Omron Sysmac Studio project MODBUS_TPC_CLIENT_NX1P2_plc_s7-1200 (Sysmac Studio 1.45.1.64010, StandardProject)

# Controller new_Controller_0: NX1P2-9024DT version 1.40
Units and slaves: Node86 : NX-ECC201 (E001); Unit 1 : NX-OD5121 (N1); Unit 2 : NX-OD4256 (N2); Unit 3 : NX-ID5342 (N3); Unit 4 : NX-ID5442 (N4); Node1 : GX-ID1611+OD16 (E002)
Task PrimaryTask (priority 4, period or condition 2000): Program0
Library OEN_Communication_V1_0_22 1.0.22 (contents left out)

VAR_GLOBAL
    NX1P2_OUT_0 : BOOL;  (* NX1P2_OUT; at BuiltInIO://cpu/#0/Output_Bit_00 *)
    NX1P2_OUT_1 : BOOL;  (* NX1P2_OUT; at BuiltInIO://cpu/#0/Output_Bit_01 *)
    NX1P2_OUT_2 : BOOL;  (* NX1P2_OUT; at BuiltInIO://cpu/#0/Output_Bit_02 *)
    NX1P2_OUT_3 : BOOL;  (* NX1P2_OUT; at BuiltInIO://cpu/#0/Output_Bit_03 *)
    NX1P2_OUT_4 : BOOL;  (* NX1P2_OUT; at BuiltInIO://cpu/#0/Output_Bit_04 *)
    NX1P2_OUT_5 : BOOL;  (* NX1P2_OUT; at BuiltInIO://cpu/#0/Output_Bit_05 *)
    NX1P2_OUT_6 : BOOL;  (* NX1P2_OUT; at BuiltInIO://cpu/#0/Output_Bit_06 *)
    NX1P2_OUT_7 : BOOL;  (* NX1P2_OUT; at BuiltInIO://cpu/#0/Output_Bit_07 *)
    NX1P2_OUT_8 : BOOL;  (* NX1P2_OUT; at BuiltInIO://cpu/#0/Output_Bit_08 *)
    NX1P2_OUT_9 : BOOL;  (* NX1P2_OUT; at BuiltInIO://cpu/#0/Output_Bit_09 *)
    GX_OUT_0 : BOOL;  (* OD_1611_DT; at ECAT://node#1/Write output 1st word/Out Bit00 *)
    GX_OUT_1 : BOOL;  (* OD_1611_DT; at ECAT://node#1/Write output 1st word/Out Bit01 *)
    GX_OUT_2 : BOOL;  (* OD_1611_DT; at ECAT://node#1/Write output 1st word/Out Bit02 *)
    GX_OUT_3 : BOOL;  (* OD_1611_DT; at ECAT://node#1/Write output 1st word/Out Bit03 *)
    GX_OUT_4 : BOOL;  (* OD_1611_DT; at ECAT://node#1/Write output 1st word/Out Bit04 *)
    GX_OUT_5 : BOOL;  (* OD_1611_DT; at ECAT://node#1/Write output 1st word/Out Bit05 *)
    GX_OUT_6 : BOOL;  (* OD_1611_DT; at ECAT://node#1/Write output 1st word/Out Bit06 *)
    GX_OUT_7 : BOOL;  (* OD_1611_DT; at ECAT://node#1/Write output 1st word/Out Bit07 *)
    GX_OUT_8 : BOOL;  (* OD_1611_DT; at ECAT://node#1/Write output 1st word/Out Bit08 *)
    GX_OUT_9 : BOOL;  (* OD_1611_DT; at ECAT://node#1/Write output 1st word/Out Bit09 *)
    GX_OUT_10 : BOOL;  (* OD_1611_DT; at ECAT://node#1/Write output 1st word/Out Bit10 *)
    GX_OUT_11 : BOOL;  (* OD_1611_DT; at ECAT://node#1/Write output 1st word/Out Bit11 *)
    GX_OUT_12 : BOOL;  (* OD_1611_DT; at ECAT://node#1/Write output 1st word/Out Bit12 *)
    GX_OUT_13 : BOOL;  (* OD_1611_DT; at ECAT://node#1/Write output 1st word/Out Bit13 *)
    GX_OUT_14 : BOOL;  (* OD_1611_DT; at ECAT://node#1/Write output 1st word/Out Bit14 *)
    GX_OUT_15 : BOOL;  (* OD_1611_DT; at ECAT://node#1/Write output 1st word/Out Bit15 *)
    REGISTER_GX_OUT : WORD;  (* OD_1611_DT; at ECAT://node#1/Write output 1st word *)
    NX1P2_IN_0 : BOOL;  (* input_nx1p2_9024dt; at BuiltInIO://cpu/#0/Input_Bit_00 *)
    NX1P2_IN_1 : BOOL;  (* input_nx1p2_9024dt; at BuiltInIO://cpu/#0/Input_Bit_01 *)
    NX1P2_IN_2 : BOOL;  (* input_nx1p2_9024dt; at BuiltInIO://cpu/#0/Input_Bit_02 *)
    NX1P2_IN_3 : BOOL;  (* input_nx1p2_9024dt; at BuiltInIO://cpu/#0/Input_Bit_03 *)
    NX1P2_IN_4 : BOOL;  (* input_nx1p2_9024dt; at BuiltInIO://cpu/#0/Input_Bit_04 *)
    NX1P2_IN_5 : BOOL;  (* input_nx1p2_9024dt; at BuiltInIO://cpu/#0/Input_Bit_05 *)
    NX1P2_IN_6 : BOOL;  (* input_nx1p2_9024dt; at BuiltInIO://cpu/#0/Input_Bit_06 *)
    NX1P2_IN_7 : BOOL;  (* input_nx1p2_9024dt; at BuiltInIO://cpu/#0/Input_Bit_07 *)
    NX1P2_IN_8 : BOOL;  (* input_nx1p2_9024dt; at BuiltInIO://cpu/#0/Input_Bit_08 *)
    NX1P2_IN_9 : BOOL;  (* input_nx1p2_9024dt; at BuiltInIO://cpu/#0/Input_Bit_09 *)
    NX1P2_IN_10 : BOOL;  (* input_nx1p2_9024dt; at BuiltInIO://cpu/#0/Input_Bit_10 *)
    NX1P2_IN_11 : BOOL;  (* input_nx1p2_9024dt; at BuiltInIO://cpu/#0/Input_Bit_11 *)
    NX1P2_IN_12 : BOOL;  (* input_nx1p2_9024dt; at BuiltInIO://cpu/#0/Input_Bit_12 *)
    NX1P2_IN_13 : BOOL;  (* input_nx1p2_9024dt; at BuiltInIO://cpu/#0/Input_Bit_13 *)
    IN_GX_0 : BOOL;  (* INPUT_ID1611; at ECAT://node#1/Read input 1st word/In Bit00 *)
    IN_GX_1 : BOOL;  (* INPUT_ID1611; at ECAT://node#1/Read input 1st word/In Bit01 *)
    IN_GX_2 : BOOL;  (* INPUT_ID1611; at ECAT://node#1/Read input 1st word/In Bit02 *)
    IN_GX_3 : BOOL;  (* INPUT_ID1611; at ECAT://node#1/Read input 1st word/In Bit03 *)
    IN_GX_4 : BOOL;  (* INPUT_ID1611; at ECAT://node#1/Read input 1st word/In Bit04 *)
    IN_GX_5 : BOOL;  (* INPUT_ID1611; at ECAT://node#1/Read input 1st word/In Bit05 *)
    IN_GX_6 : BOOL;  (* INPUT_ID1611; at ECAT://node#1/Read input 1st word/In Bit06 *)
    IN_GX_7 : BOOL;  (* INPUT_ID1611; at ECAT://node#1/Read input 1st word/In Bit07 *)
    IN_GX_8 : BOOL;  (* INPUT_ID1611; at ECAT://node#1/Read input 1st word/In Bit08 *)
    IN_GX_9 : BOOL;  (* INPUT_ID1611; at ECAT://node#1/Read input 1st word/In Bit09 *)
    IN_GX_10 : BOOL;  (* INPUT_ID1611; at ECAT://node#1/Read input 1st word/In Bit10 *)
    IN_GX_11 : BOOL;  (* INPUT_ID1611; at ECAT://node#1/Read input 1st word/In Bit11 *)
    IN_GX_12 : BOOL;  (* INPUT_ID1611; at ECAT://node#1/Read input 1st word/In Bit12 *)
    IN_GX_13 : BOOL;  (* INPUT_ID1611; at ECAT://node#1/Read input 1st word/In Bit13 *)
    IN_GX_14 : BOOL;  (* INPUT_ID1611; at ECAT://node#1/Read input 1st word/In Bit14 *)
    IN_GX_15 : BOOL;  (* INPUT_ID1611; at ECAT://node#1/Read input 1st word/In Bit15 *)
    REGISTER_IN_GX : WORD;  (* INPUT_ID1611; at ECAT://node#1/Read input 1st word *)
    ERROR_GX : BYTE;  (* INPUT_ID1611; at ECAT://node#1/Sysmac Error Status *)
END_VAR
VAR_GLOBAL RETAIN
    D0 AT %D0 : INT;
    D1 AT %D1 : INT;
    D2 AT %D2 : INT;
    D3 AT %D3 : INT;
END_VAR
VAR_GLOBAL
    W0 AT %W0 : INT;
END_VAR

PROGRAM Program0
VAR
    DISCONNECT_TCP_CLIENT : BOOL;
    TCP_CLIENT_CONNECT : BOOL;
    T_CONNECT_TCP : TON;
    T_CONNECT_TCP_CLIENT : TON;
    MODBUS_CLIENT : OEN\Modbus\ModbusTCP_Client;
    REQUEST_CLIENT : ARRAY[0..3] OF OEN\Modbus\sModbusReq := [(Enable := True, NodeAdr := 0, FunctionCode := Fn03_ReadHoldingRegisters, Read := (StartAddressRemote := 0, StartAddressLocal := 0, Count := 4), Write := (StartAddressRemote := 0, StartAddressLocal := 0, Count := 0)), (Enable := True, NodeAdr := 0, FunctionCode := Fn16_WriteMultipleRegisters, Read := (StartAddressRemote := 0, StartAddressLocal := 0, Count := 0), Write := (StartAddressRemote := 4, StartAddressLocal := 4, Count := 6)), (Enable := True, NodeAdr := 0, FunctionCode := Fn03_ReadHoldingRegisters, Read := (StartAddressRemote := 10, StartAddressLocal := 10, Count := 6), Write := (StartAddressRemote := 0, StartAddressLocal := 0, Count := 0)), (Enable := True, NodeAdr := 0, FunctionCode := Fn16_WriteMultipleRegisters, Read := (StartAddressRemote := 0, StartAddressLocal := 0, Count := 0), Write := (StartAddressRemote := 17, StartAddressLocal := 17, Count := 6))];
    DATA_COIL_CLIENT : ARRAY[0..16] OF BOOL;
    DISCRETELINPUT_CLIENT : ARRAY[0..16] OF BOOL;
    INPUT_REGISTER_CLIENT : ARRAY[0..16] OF WORD;
    HOLDINGREGISTERR_CLIENT : ARRAY[0..31] OF WORD;
    REQUEST_DONE : BOOL;
    REQUEST_CLYCLE_TIME : TIME;
    TCP_CONNECT : BOOL;
    DATA_WRITE_0 : WORD;
    DATA_WRITE_1 : WORD;
    DATA_WRITE_2 : WORD;
    DATA_WRITE_3 : WORD;
    DATA_WRITE_4 AT %W0 : WORD;
    DATA_WRITE_5 : WORD;
    INT_DATA_WRITE_5 : INT;
    INT_WRITE_4 : INT;
    DINT_DATA_WRITE_6 : DINT;
    INT_DATA_READ_4 : INT;
    INT_DATA_READ_0 : INT;
    INT_DATA_READ_1 : DINT;
    INT_DATA_READ_5 : INT;
    INT_DATA_READ_6 : INT;
    INT_DATA_LOW_READ_5 : INT;
    INT_DATA_HIGH_READ_5 : INT;
    INT_DATA_READ_7 : INT;
    DISCONNECT_MODBUS_TCP_CLIENT : BOOL;
    VAL_CONTROL_OD1611 : DWORD;
    VAL_TRGIAN_RES_01 : WORD;
    INT_DATA_CONTROL : DINT;
    INT_HIGH_RES_DWORD_0 : DINT;
    OUT : BOOL;
    DATA_READ_12 : WORD;
    DATA_READ_13 : WORD;
    REGISTER_12 : DINT;
    T_COUNT_1 : TON;
    DATA_READ_4 : WORD;
    COUNT_1 : INT;
END_VAR
VAR RETAIN
    SV_COUNT_1 : int;
END_VAR
VAR
    T_COUNT_2 : TON;
    H : INT;
END_VAR
VAR RETAIN
    DATA_RES_15 AT %D15 : WORD;
END_VAR
VAR
    T1 : TON;
    T2 : TON;
END_VAR
VAR_EXTERNAL
    REGISTER_GX_OUT : WORD;
    NX1P2_IN_0 : BOOL;
    IN_GX_0 : BOOL;
    NX1P2_OUT_3 : BOOL;
    IN_GX_1 : BOOL;
    IN_GX_2 : BOOL;
    D0 : INT;
    IN_GX_3 : BOOL;
    D1 : INT;
    IN_GX_4 : BOOL;
    D2 : INT;
    D3 : INT;
    NX1P2_OUT_5 : BOOL;
    IN_GX_6 : BOOL;
END_VAR
VAR
    _e1 : R_TRIG;
    _e2 : R_TRIG;
    _e3 : R_TRIG;
    _e4 : R_TRIG;
    _e5 : R_TRIG;
    _e6 : R_TRIG;
    _e7 : R_TRIG;
END_VAR

(* Section modbus_tcp_client: ladder, written here as Structured Text *)

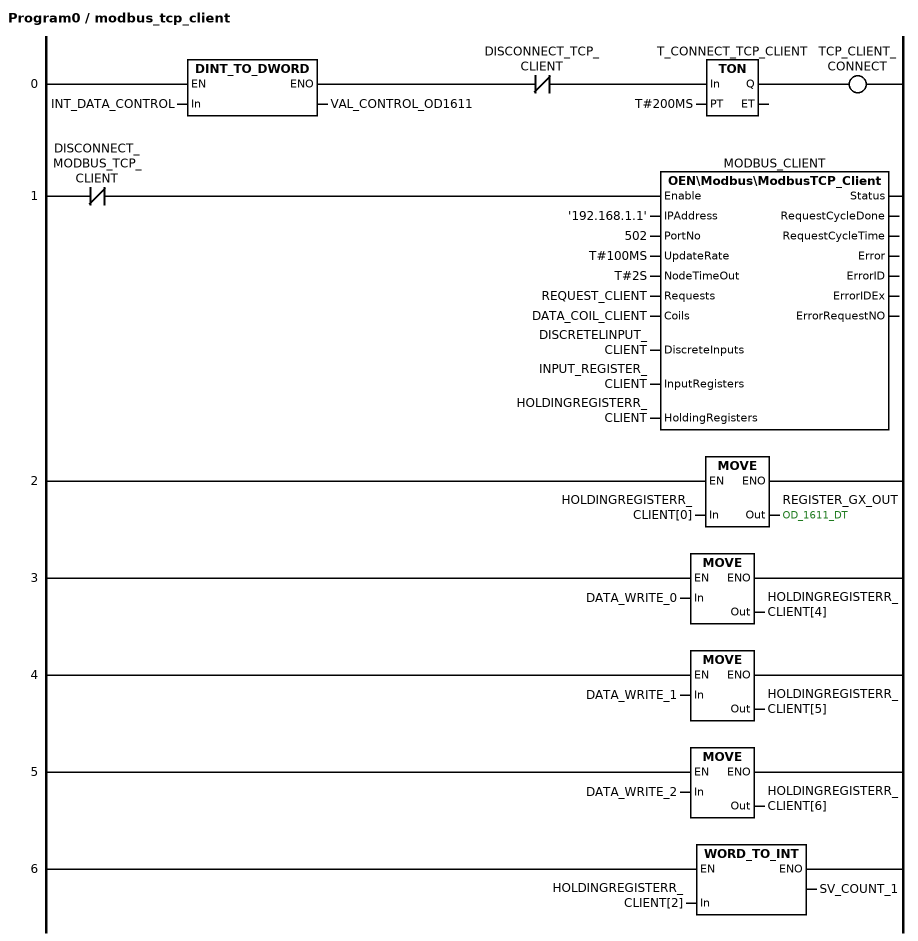
(* Rung 0 *)
VAL_CONTROL_OD1611 := DINT_TO_DWORD(In := INT_DATA_CONTROL);
T_CONNECT_TCP_CLIENT(In := NOT DISCONNECT_TCP_CLIENT, PT := T#200MS);
TCP_CLIENT_CONNECT := T_CONNECT_TCP_CLIENT.Q;
(* Rung 1 *)
MODBUS_CLIENT(Enable := NOT DISCONNECT_MODBUS_TCP_CLIENT, IPAddress := '192.168.1.1', PortNo := 502, UpdateRate := T#100MS, NodeTimeOut := T#2S, Requests := REQUEST_CLIENT, Coils := DATA_COIL_CLIENT, DiscreteInputs := DISCRETELINPUT_CLIENT, InputRegisters := INPUT_REGISTER_CLIENT, HoldingRegisters := HOLDINGREGISTERR_CLIENT);
(* Rung 2 *)
REGISTER_GX_OUT := HOLDINGREGISTERR_CLIENT[0];
(* Rung 3 *)
HOLDINGREGISTERR_CLIENT[4] := DATA_WRITE_0;
(* Rung 4 *)
HOLDINGREGISTERR_CLIENT[5] := DATA_WRITE_1;
(* Rung 5 *)
HOLDINGREGISTERR_CLIENT[6] := DATA_WRITE_2;
(* Rung 6 *)
SV_COUNT_1 := WORD_TO_INT(In := HOLDINGREGISTERR_CLIENT[2]);

(* Section write_data_res_4_10: ladder, written here as Structured Text *)

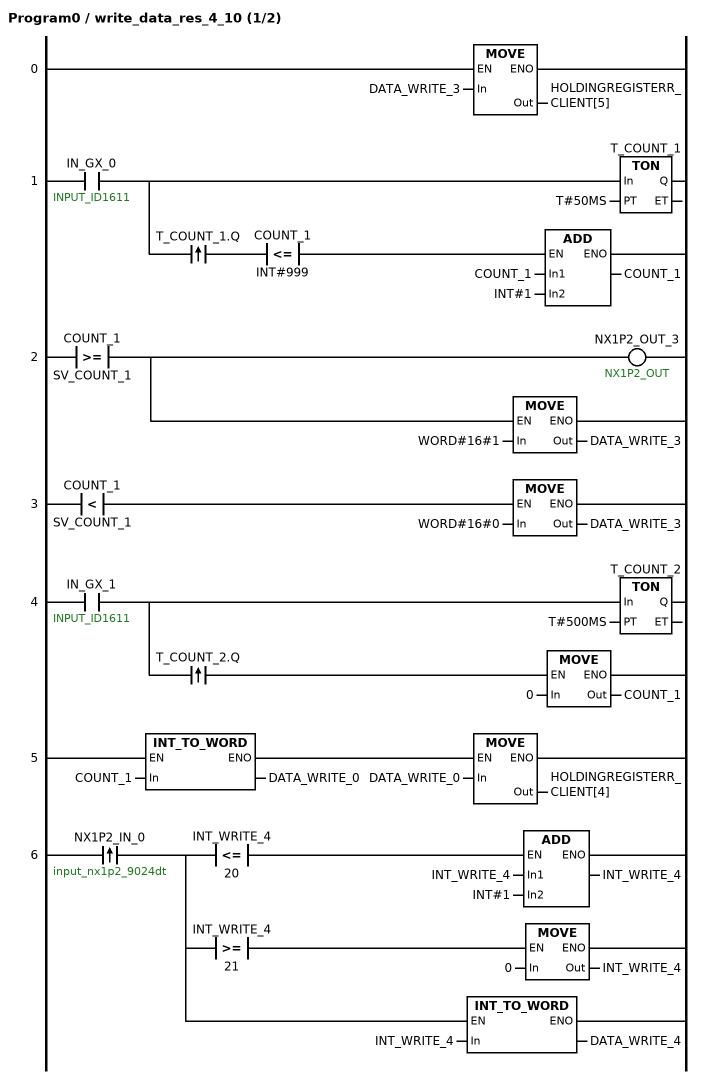
(* Rung 0 *)
HOLDINGREGISTERR_CLIENT[5] := DATA_WRITE_3;
(* Rung 1 *)
T_COUNT_1(In := IN_GX_0, PT := T#50MS);
_e1(CLK := T_COUNT_1.Q);
IF IN_GX_0 AND _e1.Q AND (COUNT_1 <= INT#999) THEN COUNT_1 := COUNT_1 + INT#1; END_IF;
(* Rung 2 *)
NX1P2_OUT_3 := COUNT_1 >= SV_COUNT_1;
IF COUNT_1 >= SV_COUNT_1 THEN DATA_WRITE_3 := WORD#16#1; END_IF;
(* Rung 3 *)
IF COUNT_1 < SV_COUNT_1 THEN DATA_WRITE_3 := WORD#16#0; END_IF;
(* Rung 4 *)
T_COUNT_2(In := IN_GX_1, PT := T#500MS);
_e2(CLK := T_COUNT_2.Q);
IF IN_GX_1 AND _e2.Q THEN COUNT_1 := 0; END_IF;
(* Rung 5 *)
DATA_WRITE_0 := INT_TO_WORD(In := COUNT_1);
HOLDINGREGISTERR_CLIENT[4] := DATA_WRITE_0;
(* Rung 6 *)
_e3(CLK := NX1P2_IN_0);
IF _e3.Q AND (INT_WRITE_4 <= 20) THEN INT_WRITE_4 := INT_WRITE_4 + INT#1; END_IF;
IF _e3.Q AND (INT_WRITE_4 >= 21) THEN INT_WRITE_4 := 0; END_IF;
IF _e3.Q THEN DATA_WRITE_4 := INT_TO_WORD(In := INT_WRITE_4); END_IF;

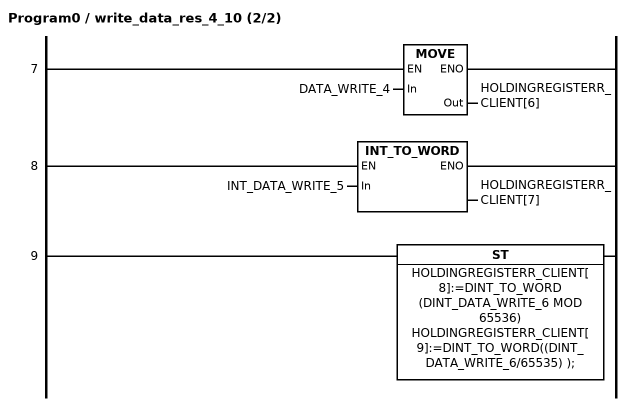
(* Rung 7 *)
HOLDINGREGISTERR_CLIENT[6] := DATA_WRITE_4;
(* Rung 8 *)
HOLDINGREGISTERR_CLIENT[7] := INT_TO_WORD(In := INT_DATA_WRITE_5);
(* Rung 9 *)
HOLDINGREGISTERR_CLIENT[8]:=DINT_TO_WORD (DINT_DATA_WRITE_6 MOD 65536);
HOLDINGREGISTERR_CLIENT[9]:=DINT_TO_WORD((DINT_DATA_WRITE_6/65535) ); 

(* Section READ_REGISTER: ladder, written here as Structured Text *)

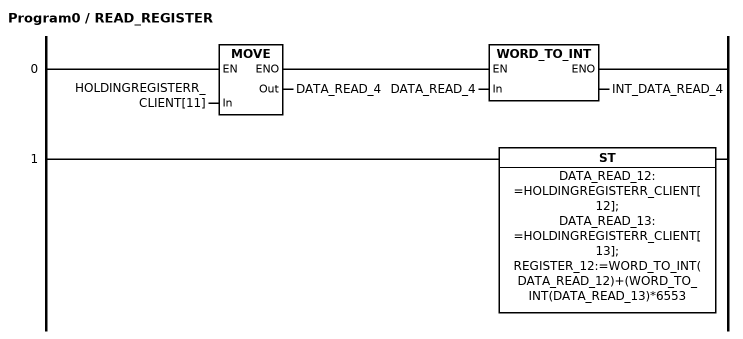
(* Rung 0 *)
DATA_READ_4 := HOLDINGREGISTERR_CLIENT[11];
INT_DATA_READ_4 := WORD_TO_INT(In := DATA_READ_4);
(* Rung 1 *)
DATA_READ_12:=HOLDINGREGISTERR_CLIENT[12];
DATA_READ_13:=HOLDINGREGISTERR_CLIENT[13];
REGISTER_12:=WORD_TO_INT(DATA_READ_12)+(WORD_TO_INT(DATA_READ_13)*65536);

(* Section REGISTER_MEMORY: ladder, written here as Structured Text *)

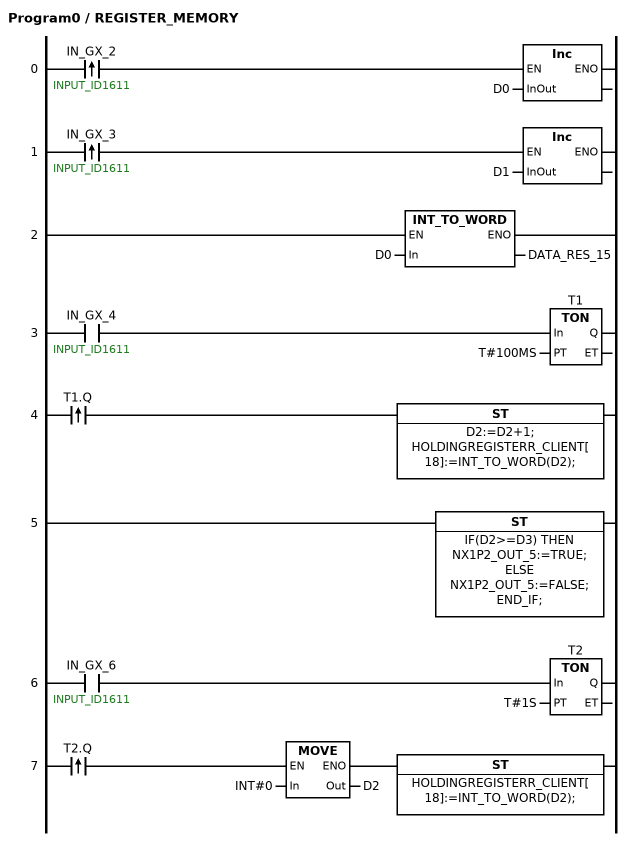
(* Rung 0 *)
_e4(CLK := IN_GX_2);
IF _e4.Q THEN Inc(InOut := D0); END_IF;
(* Rung 1 *)
_e5(CLK := IN_GX_3);
IF _e5.Q THEN Inc(InOut := D1); END_IF;
(* Rung 2 *)
DATA_RES_15 := INT_TO_WORD(In := D0);
(* Rung 3 *)
T1(In := IN_GX_4, PT := T#100MS);
(* Rung 4 *)
_e6(CLK := T1.Q);
IF _e6.Q THEN
    D2:=D2+1;
    HOLDINGREGISTERR_CLIENT[18]:=INT_TO_WORD(D2);
END_IF;
(* Rung 5 *)
IF(D2>=D3) THEN
	NX1P2_OUT_5:=TRUE;
ELSE
	NX1P2_OUT_5:=FALSE;
END_IF;
(* Rung 6 *)
T2(In := IN_GX_6, PT := T#1S);
(* Rung 7 *)
_e7(CLK := T2.Q);
IF _e7.Q THEN D2 := INT#0; END_IF;
IF _e7.Q THEN
    HOLDINGREGISTERR_CLIENT[18]:=INT_TO_WORD(D2);
END_IF;

(* Section READ_WRITE_DATA: ladder, written here as Structured Text *)

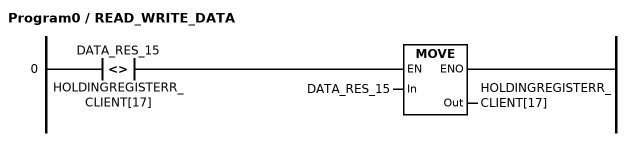
(* Rung 0 *)
IF DATA_RES_15 <> HOLDINGREGISTERR_CLIENT[17] THEN HOLDINGREGISTERR_CLIENT[17] := DATA_RES_15; END_IF;
END_PROGRAM